PROGRAM P_Palletizing
VAR CONSTANT
	cNumberOfConveyors	:INT:=6;
END_VAR

VAR
	bfull :BOOL;
	bStartInfeed :BOOL;
	fb_PickManipulator	:FB_PickManipulator;
	fbConveyor 			:ARRAY [0..cNumberOfConveyors-1] 	OF FB_Conveyor;			// Tehdään const
	convhandshake		:ARRAY [0..cNumberOfConveyors] 		OF ST_HMIHandShake;		// HMI:lle tiedonvaihto. Viimeinen on tyhjä
	//testbutton			:ARRAY [0..3] OF stTestiSeq;
	
	(*HandShake 			:(	Empty,													// Lokaali enumeraatio 
							InFeedWithForklif, 
							InFeedMiddle, 
							InFeedUnloading,
							OutFeedLoading,
							OutFeedMiddle,
							OutFeedWithForklif
							); *)
END_VAR

A_Interlocks();
A_MovementAlarms();

fb_PickManipulator(
	iostHMISequenceCtrl		:= HMI.stSeqControls[E_Stations.Portal] , 
	                    	
	ioAxis					:= IO.ServoAxis, 
	ioAxisHMI				:= HMI.parServoAxis, 
	iostRobotCom			:= gFeeding.stRobotCom, 
	istMachineStates		:= HMI.stMachineStates[E_Stations.Portal] , 
	istPositionParameters	:= HMI.parManipulator,
 
	ibPalletInPos10			:= JTA.fbSensor[SEN_10S3_Lava_kuljettimella_3].oState,
	ibPalletInPos11			:= JTA.fbSensor[SEN_11S3_Lava_kuljettimella_3].oState, 
	ibVacuumON_1			:= JTA.fbSensor[SEN_70B1_Alipaineen_tunnistus_1].oState,
	ibVacuumON_2			:= JTA.fbSensor[SEN_70B2_Alipaineen_tunnistus_2].oState, 
	ibCollisionDetection	:= JTA.fbSensor[SEN_70S5_Tormaysraja_1].oState, 
	ibClampOpenLeft			:= JTA.fbSensor[SEN_70S2_Manipulaattori_kynnet_auki_1].oState, 
	ibClampCloseLeft		:= JTA.fbSensor[SEN_70S1_Manipulaattori_kynnet_kiinni_1].oState, 
	ibClampOpenRight		:= JTA.fbSensor[SEN_70S4_Manipulaattori_kynnet_auki_2].oState, 
	ibClampCloseRight		:= JTA.fbSensor[SEN_70S3_Manipulaattori_kynnet_kiinni_2].oState, 
	
	obCloseClamps			=> JTA.fbCylinders[VEN_70V1_Manipulaattori_kynnet_kiinni].iDriveOutCW, 
	obOpenClamps			=> JTA.fbCylinders[VEN_70V1_Manipulaattori_kynnet_kiinni].iDriveInCCW, 
	obVacuumOn				=> JTA.fbCylinders[VEN_70V2_Ejektori_imu].iDriveOutCW, 
	oError					=> , 
	oErrorID				=> );


gfeeding.fbAxisCMMT[E_Axis.AXEN_70M1_X_VAAKALIIKE](
	ioAxis				:= IO.ServoAxis[E_Axis.AXEN_70M1_X_VAAKALIIKE], 
	ioHMI				:= HMI.parServoAxis[E_Axis.AXEN_70M1_X_VAAKALIIKE], 
	iMachineState		:= HMI.stMachineStates[E_Stations.Portal], 
	iOverride			:= HMI.Overrdive[E_Stations.Portal] );	

gfeeding.fbAxisCMMT[E_Axis.AXEN_70M2_Z_PYSTYLIIKE](
	ioAxis				:= IO.ServoAxis[E_Axis.AXEN_70M2_Z_PYSTYLIIKE], 
	ioHMI				:= HMI.parServoAxis[E_Axis.AXEN_70M2_Z_PYSTYLIIKE], 
	iMachineState		:= HMI.stMachineStates[E_Stations.Portal], 
	iOverride			:= HMI.Overrdive[E_Stations.Portal] );	
	
// ************************ Kuljetinohjaukset ****************************
{region "Conveyor control"}

//IbStopSensor käynnistää ekan kuljettimen!
//Käynnistysehdot ekalle syöttökuljettimelle: 
//-Nappikotelon startin liipaisu (Ajon eka lava)
//-Viimeisellä kuljettimella lava ja ekalle nostetaan lava. Tässä syytä laittaa sensoriin viivettä tarpeeksi Visun kautta! 
bStartInfeed := JTA.fbSensor[SEN_100BB1_Start_nappi].oState;// OR (JTA.fbSensor[SEN_10S3_Lava_kuljettimella_3].oState AND JTA.fbSensor[SEN_10S1_Lava_kuljettimella_1].oState); 
		  
fbConveyor[E_Conveyor.InFeedWithForklif](
	iostHMISequenceCtrl		:= HMI.stSeqControls[E_Stations.Feeding]  , 
	PreviousHandshake		:= convhandshake[E_Conveyor.InFeedWithForklif], 
	NextHandshake			:= convhandshake[E_Conveyor.InFeedMiddle], 
	ibStopSensor			:= bStartInfeed,//JTA.fbSensor[SEN_10S1_Lava_kuljettimella_1].oState, 
	ibNextVFDRunning		:= HMI.parABB380[E_VFDControls.VDFEN_10M2_Syottokuljetin].ledMoving.State,			// Tähän tamun käy tieto seuraavalta kuljettimelta
	ibProcessingFinnished	:= TRUE,
	oStartConveyor		=> IO.fbSEWMovimot[E_VFDControls.VDFEN_10M1_Syottokuljetin].iStart);
	

fbConveyor[E_Conveyor.InFeedMiddle](
	iostHMISequenceCtrl		:= HMI.stSeqControls[E_Stations.Feeding]  , 
	PreviousHandshake		:= convhandshake[E_Conveyor.InFeedMiddle], 
	NextHandshake			:= convhandshake[E_Conveyor.InFeedUnloading], 
	ibStopSensor			:= JTA.fbSensor[SEN_10S2_Lava_kuljettimella_2].oState, 
	ibNextVFDRunning		:= HMI.parABB380[E_VFDControls.VDFEN_10M3_Syottokuljetin].ledMoving.State,		// Tähän tamun käy tieto seuraavalta kuljettimelta
	ibProcessingFinnished	:= TRUE,

	oStartConveyor		=> IO.fbSEWMovimot[E_VFDControls.VDFEN_10M2_Syottokuljetin].iStart);
	
fbConveyor[E_Conveyor.InFeedUnloading](
	iostHMISequenceCtrl		:= HMI.stSeqControls[E_Stations.Feeding], 
	PreviousHandshake		:= convhandshake[E_Conveyor.InFeedUnloading], 
	NextHandshake			:= convhandshake[E_Conveyor.Empty], 
	ibStopSensor			:= JTA.fbSensor[SEN_10S3_Lava_kuljettimella_3].oState, 
	ibNextVFDRunning		:= FALSE,		// Tähän tamun käy tieto seuraavalta kuljettimelta
	ibProcessingFinnished	:= TRUE,
	oStartConveyor		=> IO.fbSEWMovimot[E_VFDControls.VDFEN_10M3_Syottokuljetin].iStart);
 

//Poistokuljettimien pyörimissuuntien käännöt
IO.fbSEWMovimot[E_VFDControls.VDFEN_11M3_Poistokuljetin].iBWD := TRUE;
IO.fbSEWMovimot[E_VFDControls.VDFEN_11M2_Poistokuljetin].iBWD := TRUE;
IO.fbSEWMovimot[E_VFDControls.VDFEN_11M1_Poistokuljetin].iBWD := TRUE;	 
	 
		  
fbConveyor[E_Conveyor.OutFeedLoading](
	iostHMISequenceCtrl	:= HMI.stSeqControls[E_Stations.Outfeeding]  , 
	PreviousHandshake	:= convhandshake[E_Conveyor.OutFeedLoading], 
	NextHandshake		:= convhandshake[E_Conveyor.OutFeedMiddle], 
	ibStopSensor		:= gFeeding.stRobotCom.PalletFull OR bfull, 
	ibNextVFDRunning	:= HMI.parABB380[E_VFDControls.VDFEN_11M2_Poistokuljetin].ledMoving.State,			// Tähän tamun käy tieto seuraavalta kuljettimelta
	ibProcessingFinnished	:= TRUE,
		 
	oStartConveyor		=> IO.fbSEWMovimot[E_VFDControls.VDFEN_11M3_Poistokuljetin].iStart);
	

fbConveyor[E_Conveyor.OutFeedMiddle](
	iostHMISequenceCtrl		:= HMI.stSeqControls[E_Stations.Outfeeding]  , 
	PreviousHandshake		:= convhandshake[E_Conveyor.OutFeedMiddle], 
	NextHandshake			:= convhandshake[E_Conveyor.OutFeedWithForklif], 
	ibStopSensor			:= JTA.fbSensor[SEN_11S2_Lava_kuljettimella_2].oState, 
	ibNextVFDRunning		:= HMI.parABB380[E_VFDControls.VDFEN_11M1_Poistokuljetin].ledMoving.State,		// Tähän tamun käy tieto seuraavalta kuljettimelta
	ibProcessingFinnished	:= TRUE,
	oStartConveyor		=>  IO.fbSEWMovimot[E_VFDControls.VDFEN_11M2_Poistokuljetin].iStart);

	
fbConveyor[E_Conveyor.OutFeedWithForklif](
	iostHMISequenceCtrl		:= HMI.stSeqControls[E_Stations.Outfeeding], 
	PreviousHandshake		:= convhandshake[E_Conveyor.OutFeedWithForklif], 
	NextHandshake			:= convhandshake[E_Conveyor.Empty], 
	ibStopSensor			:= JTA.fbSensor[SEN_11S1_Lava_kuljettimella_1].oState, 
	ibNextVFDRunning		:= FALSE,		// Tähän tamun käy tieto seuraavalta kuljettimelta
	ibProcessingFinnished	:= TRUE,
	oStartConveyor		=> IO.fbSEWMovimot[E_VFDControls.VDFEN_11M1_Poistokuljetin].iStart);
		  
			   
{endregion}
// ************************ Kuljetinohjaukset ****************************

ACTION A_Interlocks:
// Servojen overdrive
JTA.fbAxisAX8000[AXEN_70M1_X_VAAKALIIKE].iOverride					:= HMI.Overrdive[E_Stations.Portal];		
JTA.fbAxisAX8000[AXEN_70M2_Z_PYSTYLIIKE].iOverride					:= HMI.Overrdive[E_Stations.Portal];		
	


//Servojen paikat testattu lukituksiin 20.8 J-MN
//Lukitukset telineen välissä ylöspäin mentäessä
gfeeding.fbAxisCMMT[AXEN_70M2_Z_PYSTYLIIKE].M_InterlockPos				(LockingON:= (IO.ServoAxis[AXEN_70M1_X_VAAKALIIKE].AxisRef.NcToPlc.ActPos < 1065 AND 
																	IO.ServoAxis[AXEN_70M2_Z_PYSTYLIIKE].AxisRef.NcToPlc.ActPos > 1370 AND 
																	IO.ServoAxis[AXEN_70M2_Z_PYSTYLIIKE].AxisRef.NcToPlc.ActPos < 1640), LockingName:= 'Törmäysvaara' );
//Lukitukset telineen välissä ja yläpuolella alaspäin mentäessä
gfeeding.fbAxisCMMT[AXEN_70M2_Z_PYSTYLIIKE].M_InterlockNeg				(LockingON:= ((	IO.ServoAxis[AXEN_70M1_X_VAAKALIIKE].AxisRef.NcToPlc.ActPos < 1100 AND
																						IO.ServoAxis[AXEN_70M1_X_VAAKALIIKE].AxisRef.NcToPlc.ActPos > 150 AND
																						IO.ServoAxis[AXEN_70M2_Z_PYSTYLIIKE].AxisRef.NcToPlc.ActPos < 1700)
																						OR
																						(IO.ServoAxis[AXEN_70M1_X_VAAKALIIKE].AxisRef.NcToPlc.ActPos < 55 AND 
																						IO.ServoAxis[AXEN_70M2_Z_PYSTYLIIKE].AxisRef.NcToPlc.ActPos < 1660) //Telineen yläpuolella
																						OR
																						(IO.ServoAxis[AXEN_70M1_X_VAAKALIIKE].AxisRef.NcToPlc.ActPos < 1100 AND 
																						IO.ServoAxis[AXEN_70M2_Z_PYSTYLIIKE].AxisRef.NcToPlc.ActPos > 1380 AND
																						IO.ServoAxis[AXEN_70M2_Z_PYSTYLIIKE].AxisRef.NcToPlc.ActPos < 1650)
																						OR 	
																						(IO.ServoAxis[AXEN_70M1_X_VAAKALIIKE].AxisRef.NcToPlc.ActPos < 1100 AND  													 	
																						IO.ServoAxis[AXEN_70M2_Z_PYSTYLIIKE].AxisRef.NcToPlc.ActPos < 1215)), LockingName:= 'Törmäysvaara' ); //Telineen välissä
//Lukitukset telineeseen päin liikuttaessa X-suunnassa
gfeeding.fbAxisCMMT[AXEN_70M1_X_VAAKALIIKE].M_InterlockNeg				(LockingON:= (IO.ServoAxis[AXEN_70M1_X_VAAKALIIKE].AxisRef.NcToPlc.ActPos < 1065 AND 
																	((IO.ServoAxis[AXEN_70M2_Z_PYSTYLIIKE].AxisRef.NcToPlc.ActPos > 1370 AND 
																	IO.ServoAxis[AXEN_70M2_Z_PYSTYLIIKE].AxisRef.NcToPlc.ActPos < 1750) OR 													 	
																	IO.ServoAxis[AXEN_70M2_Z_PYSTYLIIKE].AxisRef.NcToPlc.ActPos < 1300)) OR //Telineen välissä telineeseenpäin	
																	IO.ServoAxis[AXEN_70M1_X_VAAKALIIKE].AxisRef.NcToPlc.ActPos < 49, LockingName:= 'Törmäysvaara' ); //Telineen takareuna																	

IO.fbSEWMovimot[VDFEN_10M3_Syottokuljetin].M_InterlockPos				(LockingON:= IO.ServoAxis[AXEN_70M2_Z_PYSTYLIIKE].AxisRef.NcToPlc.ActPos < 1500 , LockingName:= 'Törmäysvaara' ); //Solun pään kuljettimet ei saa liikkua jos manipulaattori liian alhaalla	
IO.fbSEWMovimot[VDFEN_10M3_Syottokuljetin].M_InterlockNeg				(LockingON:= IO.ServoAxis[AXEN_70M2_Z_PYSTYLIIKE].AxisRef.NcToPlc.ActPos < 1500 , LockingName:= 'Törmäysvaara' ); //Solun pään kuljettimet ei saa liikkua jos manipulaattori liian alhaalla
IO.fbSEWMovimot[VDFEN_11M3_Poistokuljetin].M_InterlockPos				(LockingON:= IO.ServoAxis[AXEN_70M2_Z_PYSTYLIIKE].AxisRef.NcToPlc.ActPos < 1500 , LockingName:= 'Törmäysvaara' ); //Solun pään kuljettimet ei saa liikkua jos manipulaattori liian alhaalla	
IO.fbSEWMovimot[VDFEN_11M3_Poistokuljetin].M_InterlockNeg				(LockingON:= IO.ServoAxis[AXEN_70M2_Z_PYSTYLIIKE].AxisRef.NcToPlc.ActPos < 1500 , LockingName:= 'Törmäysvaara' ); //Solun pään kuljettimet ei saa liikkua jos manipulaattori liian alhaalla																
	

															
// Sulake viimeinen
//JTA.fbAxisAX8000[AXEN_70M1_X_VAAKALIIKE].M_InterlockNeg			(NOT JTA.fbSensor[SEN_20F1_Servovahvistin_sulake_NOK].oState, 'Sulake 20F1');
//JTA.fbAxisAX8000[AXEN_70M1_X_VAAKALIIKE].M_InterlockPos			(NOT JTA.fbSensor[SEN_20F1_Servovahvistin_sulake_NOK].oState, 'Sulake 20F1');
//JTA.fbAxisAX8000[AXEN_70M2_Z_PYSTYLIIKE].M_InterlockNeg			(NOT JTA.fbSensor[SEN_20F1_Servovahvistin_sulake_NOK].oState, 'Sulake 20F1');
//JTA.fbAxisAX8000[AXEN_70M2_Z_PYSTYLIIKE].M_InterlockPos			(NOT JTA.fbSensor[SEN_20F1_Servovahvistin_sulake_NOK].oState, 'Sulake 20F1');


// Sylintereiden lukitukset
//JTA.fbCylinders[VEN_20Y1_Leuka_avaus].M_InterlockPos				(NOT JTA.fbSensor[SEN_110S1_Painekytkin].oState, 'Paineilma alhainen');	
//JTA.fbCylinders[VEN_20Y1_Leuka_avaus].M_InterlockNeg				(NOT JTA.fbSensor[SEN_110S1_Painekytkin].oState, 'Paineilma alhainen');			

// Tamun lukitukset
//IO.fbABB380[VDFEN_60M1_KAANTOMANIPULAATTORI].M_InterlockPos(NOT JTa.fbSensor[SEN_61S1_Luisti_takana_10].oState,concat('Anturi: ',HMI.parSensor[SEN_61S1_Luisti_takana_10].DeviceData.btnName));


// MACHINE STATES 	

JTA.fbCylinders[VEN_70V1_Manipulaattori_kynnet_kiinni].iMachineState:= HMI.stMachineStates[E_Stations.Portal];	
JTA.fbCylinders[VEN_70V2_Ejektori_imu].iMachineState				:= HMI.stMachineStates[E_Stations.Portal];	

 
JTA.fbAxisAX8000[AXEN_70M1_X_VAAKALIIKE].iMachineState				:= HMI.stMachineStates[E_Stations.Portal];		
JTA.fbAxisAX8000[AXEN_70M2_Z_PYSTYLIIKE].iMachineState				:= HMI.stMachineStates[E_Stations.Portal];

IO.fbSEWMovimot[VDFEN_10M1_Syottokuljetin].iMachineState			:= HMI.stMachineStates[E_Stations.Portal];
IO.fbSEWMovimot[VDFEN_10M2_Syottokuljetin].iMachineState			:= HMI.stMachineStates[E_Stations.Portal];
IO.fbSEWMovimot[VDFEN_10M3_Syottokuljetin].iMachineState			:= HMI.stMachineStates[E_Stations.Portal];

IO.fbSEWMovimot[VDFEN_11M1_Poistokuljetin].iMachineState			:= HMI.stMachineStates[E_Stations.Portal];
IO.fbSEWMovimot[VDFEN_11M2_Poistokuljetin].iMachineState			:= HMI.stMachineStates[E_Stations.Portal];
IO.fbSEWMovimot[VDFEN_11M3_Poistokuljetin].iMachineState			:= HMI.stMachineStates[E_Stations.Portal];
END_ACTION

ACTION A_MovementAlarms:
// Liikeaika hälytykset 
JTA.fbSensor[SEN_70B1_Alipaineen_tunnistus_1].MovementInput			:=JTA.fbCylinders[VEN_70V2_Ejektori_imu].oPistonOutOrCW;
JTA.fbSensor[SEN_70B2_Alipaineen_tunnistus_2].MovementInput			:=JTA.fbCylinders[VEN_70V2_Ejektori_imu].oPistonOutOrCW;


JTA.fbSensor[SEN_70S1_Manipulaattori_kynnet_kiinni_1].MovementInput	:=JTA.fbCylinders[VEN_70V1_Manipulaattori_kynnet_kiinni].oPistonOutOrCW;
JTA.fbSensor[SEN_70S3_Manipulaattori_kynnet_kiinni_2].MovementInput	:=JTA.fbCylinders[VEN_70V1_Manipulaattori_kynnet_kiinni].oPistonOutOrCW;

JTA.fbSensor[SEN_70S2_Manipulaattori_kynnet_auki_1].MovementInput	:=JTA.fbCylinders[VEN_70V1_Manipulaattori_kynnet_kiinni].oPistonInCCW;
JTA.fbSensor[SEN_70S4_Manipulaattori_kynnet_auki_2].MovementInput	:=JTA.fbCylinders[VEN_70V1_Manipulaattori_kynnet_kiinni].oPistonInCCW;
END_ACTION

END_PROGRAM

(* stored: Version 1.1.0.1, ProductVersion 3.1.4024.10
   POU P_Palletizing: Id {8dddb4f8-4f55-4270-b1bb-134050f406f6}, SpecialFunc None
   Action A_Interlocks: Id {1d4a8fad-466d-4d3d-a28c-aae6a2f5acc2}
   Action A_MovementAlarms: Id {313cb909-2ad8-4c7b-8198-ee7b1a79de72} *)
